(* CoDeSys 2.3 export: GLOBAL_VARIABLES.EXP *)

(* Global variable list: Global_Variables *)
VAR_GLOBAL
	K14PumpFaulty : ARRAY [1..MAX_K14_PUMPS_NUM] OF BOOL;
	(*Неиправен 1-3 насос группы К14?*)

	K15PumpFaulty : ARRAY [1..MAX_K15_PUMPS_NUM] OF BOOL;
	(*Неиправен 1-3 насос группы К16?*)

	K16PumpFaulty : ARRAY [1..MAX_K16_PUMPS_NUM] OF BOOL;
	(*Неиправен 1-3 насос группы К16?*)
END_VAR
